Messenger.OnCondition(inoIoData.AcquisitionStatus.OfflineReason0 AND _onlineTimer.Q).Info('<#Camera offline:The vision system$'s job is being modified.#>');
Messenger.OnCondition(inoIoData.AcquisitionStatus.OfflineReason0 AND _onlineTimer.Q).Info('<#Camera offline:A discrete signal is holding the vision system Offline.#>');
Messenger.OnCondition(inoIoData.AcquisitionStatus.OfflineReason0 AND _onlineTimer.Q).Info('<#Camera offline:A communications protocol is holding the vision system Offline.#>');
END_METHOD

METHOD INTERNAL InvalidReference : BOOL
InvalidReference := FALSE;
IF NOT __ISVALIDREF(inoIoData) THEN
	_varInfo :=__VARINFO(inoIoData);
	Messenger.Programming(_sb.Clear().Append('<#Invalid reference: #>').Append(_varInfo.Symbol).ToString());
    InvalidReference := TRUE;
END_IF
END_METHOD

PROPERTY LastResultData : TcoInsightResults_v_5_x_x
GET
LastResultData := THIS^._results;
END_GET
END_PROPERTY

(*~
	<docu>
		<summary>
			Restores this instance to the Ready state. Can be called explicitly or from within one of the restore mechanisms.	
		</summary>			
	</docu>	
~*)
METHOD Restore : ITcoRestorable
_updateSignalStatesTask.Restore();
_changeJobByNumberTask.Restore();
_changeJobByNameTask.Restore();
_clearInspectionResultsTask.Restore();
_softEventTask.Restore();
_triggerTask.Restore();
_clearUserDataTask.Restore();
_setUserDataTask.Restore();

Tc2_System.MEMSET(destAddr:= ADR(THIS^._results.InspectionResults) , fillByte:= 0 , n:= SIZEOF(THIS^._results.InspectionResults));
Tc2_System.MEMSET(destAddr:= ADR(THIS^._userData.UserData) , fillByte:= 0 , n:= SIZEOF(THIS^._userData.UserData));


THIS^._results.InspectionId := 0;
THIS^._results.ResultCode := 0;
	
IF InvalidReference() THEN
    RETURN;
END_IF

Tc2_System.MEMSET(destAddr:= ADR(THIS^.inoIoData) , fillByte:= 0 , n:= SIZEOF(THIS^.inoIoData));

_status.ActionDescription := '<#Restore executed!#>';
_restoreTask.Restore();
END_METHOD

(*~
	<docu>
		<summary>
		    Custom service (manual, maintenance) logic.
			This method must be implemented in derived class.
		</summary>			
	</docu>	
~*)
METHOD PROTECTED ServiceMode
END_METHOD

(*~
	<docu>
		<summary>
			Set user data. 		
		</summary>			
	</docu>	
~*)
METHOD SetUserData : TcoCore.ITcoTaskStatus
SetUserData := THIS^._setUserDataTask.Invoke();
END_METHOD

METHOD SetUserDataAsByte : BOOL;
VAR_INPUT
	inValue : BYTE;
	inPosition : UINT;	
END_VAR
VAR
	_bufferSize : UINT; 
	_size : UINT; 
END_VAR
SetUserDataAsByte := FALSE;

_size := SIZEOF(inValue);

_bufferSize := SIZEOF(THIS^._userData.UserData)/SIZEOF(THIS^._userData.UserData[0]);

IF (inPosition +_size) > THIS^._config.UserDataSize THEN
	Messenger.Info('<#Index of UserData in method SetUserDataAsByte exceeds the size hardware structure mapped#>');
	RETURN;
END_IF

IF (inPosition +_size) > _bufferSize THEN
	Messenger.Info('<#Index of UserData in method SetUserDataAsByte exceeds the defined size#>');
	RETURN;
END_IF

THIS^._userData.UserData[inPosition]:=inValue;

SetUserDataAsByte := TRUE;
END_METHOD

METHOD SetUserDataAsDint : BOOL
VAR_INPUT
	inValue : DINT;
	inPosition : UINT;	
END_VAR
VAR
	_index : UINT;
	_size : UINT;
	_bufferSize : UINT; 
END_VAR
SetUserDataAsDint := FALSE;

_size := SIZEOF(inValue);

_bufferSize := SIZEOF(THIS^._userData.UserData)/SIZEOF(THIS^._userData.UserData[0]);

IF (inPosition +_size) > THIS^._config.UserDataSize THEN
	Messenger.Info('<#Index of UserData in method SetUserDataAsDint exceeds the size hardware structure mapped#>');
	RETURN;
END_IF

IF (inPosition +_size) > _bufferSize THEN
	Messenger.Info('<#Index of UserData in method SetUserDataAsDint exceeds the defined size#>');
	RETURN;
END_IF

TcoDintToBytes(THIS^._config.DataFormat,
				inValue,
				_userData.UserData[inPosition],
				_userData.UserData[inPosition+1],
				_userData.UserData[inPosition+2],
				_userData.UserData[inPosition+3]);	

SetUserDataAsDint := TRUE;
END_METHOD

METHOD SetUserDataAsReal : BOOL
VAR_INPUT
	inValue : DINT;
	inPosition : UINT;	
END_VAR
VAR
	_index : UINT;
	_size : UINT;
	_bufferSize : UINT; 
END_VAR
SetUserDataAsReal := FALSE;

_size := SIZEOF(inValue);

_bufferSize := SIZEOF(THIS^._userData.UserData)/SIZEOF(THIS^._userData.UserData[0]);

IF (inPosition +_size) > THIS^._config.UserDataSize THEN
	Messenger.Info('<#Index of UserData in method SetUserDataAsReal exceeds the size hardware structure mapped#>');
	RETURN;
END_IF

IF (inPosition +_size) > _bufferSize THEN
	Messenger.Info('<#Index of UserData in method SetUserDataAsReal exceeds the defined size#>');
	RETURN;
END_IF

	
TcoRealToBytes(THIS^._config.DataFormat,
				inValue,
				_userData.UserData[inPosition],
				_userData.UserData[inPosition+1],
				_userData.UserData[inPosition+2],
				_userData.UserData[inPosition+3]);			

SetUserDataAsReal := TRUE;
END_METHOD

METHOD SetUserDataAsString : BOOL
VAR_INPUT
	inValue : STRING;
	inPosition : UINT;	
END_VAR
VAR
	_index : UINT;
	_size : UINT;
	_bufferSize : UINT; 
END_VAR
SetUserDataAsString := FALSE;

_size := LEN(inValue);

_bufferSize := SIZEOF(THIS^._userData.UserData)/SIZEOF(THIS^._userData.UserData[0]);

IF (inPosition +_size) > THIS^._config.UserDataSize THEN
	Messenger.Info('<#Index of UserData in method SetUserDataAsString exceeds the size hardware structure mapped#>');
	RETURN;
END_IF

IF (inPosition +_size) > _bufferSize THEN
	Messenger.Info('<#Index of UserData in method SetUserDataAsString exceeds the defined size#>');
	RETURN;
END_IF

FOR	_index := 1 TO _size BY 1 DO	
	_userData.UserData[inPosition + _index-1] := F_ToASC(MID(inValue,1,_index));
END_FOR;

FOR	_index := inPosition +_size TO _bufferSize BY 1 DO	
	_userData.UserData[_index] := 0;
END_FOR;

SetUserDataAsString := TRUE;
END_METHOD

(*~
	<docu>
		<summary>
			Gets the `SetUserDataTask` task that controls to set of the user data. 		
		</summary>			
	</docu>	
~*)
PROPERTY SetUserDataTask : TcoCore.ITcoTaskStatus
GET
SetUserDataTask := THIS^._setUserDataTask;
END_GET
END_PROPERTY

(*~
	<docu>
		<summary>
			Executes the soft event. 		
		</summary>			
	</docu>	
~*)
METHOD SoftEvent : TcoCore.ITcoTaskStatus
VAR_INPUT
    inSoftEventNumber : UINT;
END_VAR
SoftEvent := THIS^._softEventTask.InvokeWithParameters(inSoftEventNumber);
END_METHOD

(*~
	<docu>
		<summary>
			Gets the `ClearResultDataTask` task that controls clearing of the results data. 		
		</summary>			
	</docu>	
~*)
PROPERTY SoftEventTask : TcoCore.ITcoTaskStatus
GET
SoftEventTask := THIS^._softEventTask;
END_GET
END_PROPERTY

(*~
	<docu>
		<summary>
			Gets the status of the sensor. 					
		</summary>			
	</docu>	
~*)
PROPERTY Status : REFERENCE TO TcoInsightStatus_v_5_x_x
GET
Status REF= _status;
END_GET
END_PROPERTY

(*~
	<docu>
		<summary>
			Triggers the reading sequence and waits for results. 		
		</summary>			
	</docu>	
~*)
METHOD Trigger : TcoCore.ITcoTaskStatus
Trigger := THIS^._triggerTask.Invoke();
END_METHOD

(*~
	<docu>
		<summary>
			Gets the `TriggerTask` result. 		
		</summary>			
	</docu>	
~*)
PROPERTY TriggerTask : TcoCore.ITcoTaskStatus
GET
TriggerTask := THIS^._triggerTask;
END_GET
END_PROPERTY

METHOD INTERNAL UpdateSignalStates
_status.SignalStatus.AcquisitionTriggerEnable := inoIoData.AcquisitionControl.AcquisitionTriggerEnable;
_status.SignalStatus.AcquisitionTrigger := inoIoData.AcquisitionControl.AcquisitionTrigger;
_status.SignalStatus.ClearExposureComplete := inoIoData.AcquisitionControl.ClearExposureComplete;
_status.SignalStatus.SetOffline := inoIoData.AcquisitionControl.SetOffline;
  
_status.SignalStatus.EnableResultsBuffering := inoIoData.InspectionControl.EnableResultsBuffering;
_status.SignalStatus.AcknowledgeInspectionResults := inoIoData.InspectionControl.AcknowledgeInspectionResults;
_status.SignalStatus.ExtendedUserDataSet := inoIoData.InspectionControl.ExtendedUserDataSet;
_status.SignalStatus.ExecuteCommand := inoIoData.InspectionControl.ExecuteCommand;
_status.SignalStatus.ClearError := inoIoData.InspectionControl.ClearError;
  
_status.SignalStatus.Command := inoIoData.CommandControl.Command;
  
_status.SignalStatus.TriggerSoftEvent.0 := inoIoData.SoftEventControl.TriggerSoftEvent[0];
_status.SignalStatus.TriggerSoftEvent.1 := inoIoData.SoftEventControl.TriggerSoftEvent[1];
_status.SignalStatus.TriggerSoftEvent.2 := inoIoData.SoftEventControl.TriggerSoftEvent[2];
_status.SignalStatus.TriggerSoftEvent.3 := inoIoData.SoftEventControl.TriggerSoftEvent[3];
_status.SignalStatus.TriggerSoftEvent.4 := inoIoData.SoftEventControl.TriggerSoftEvent[4];
_status.SignalStatus.TriggerSoftEvent.5 := inoIoData.SoftEventControl.TriggerSoftEvent[5];
_status.SignalStatus.TriggerSoftEvent.6 := inoIoData.SoftEventControl.TriggerSoftEvent[6];
_status.SignalStatus.TriggerSoftEvent.7 := inoIoData.SoftEventControl.TriggerSoftEvent[7];
	
_status.SignalStatus.AcquisitionTriggerReady := inoIoData.AcquisitionStatus.AcquisitionTriggerReady;
_status.SignalStatus.AcquisitionTriggerAcknowledge := inoIoData.AcquisitionStatus.AcquisitionTriggerAcknowledge;
_status.SignalStatus.ExposureComplete := inoIoData.AcquisitionStatus.ExposureComplete;
_status.SignalStatus.MissedAcquisition := inoIoData.AcquisitionStatus.MissedAcquisition;
_status.SignalStatus.OfflineReason0 := inoIoData.AcquisitionStatus.OfflineReason0;
_status.SignalStatus.OfflineReason1 := inoIoData.AcquisitionStatus.OfflineReason1;
_status.SignalStatus.OfflineReason2 := inoIoData.AcquisitionStatus.OfflineReason2;
_status.SignalStatus.Online := inoIoData.AcquisitionStatus.Online;
_status.SignalStatus.AcquisitionID := inoIoData.AcquisitionStatus.AcquisitionID;

_status.SignalStatus.SystemBusy := inoIoData.InspectionStatus.SystemBusy;
_status.SignalStatus.InspectionCompleted := inoIoData.InspectionStatus.InspectionCompleted;
_status.SignalStatus.ResultsBufferOverrun := inoIoData.InspectionStatus.ResultsBufferOverrun;
_status.SignalStatus.ResultsValid := inoIoData.InspectionStatus.ResultsValid;
_status.SignalStatus.CommandExecuting := inoIoData.InspectionStatus.CommandExecuting;
_status.SignalStatus.CommandComplete := inoIoData.InspectionStatus.CommandComplete;
_status.SignalStatus.CommandFailed := inoIoData.InspectionStatus.CommandFailed;
_status.SignalStatus.ExtendedUserDataSetAcknowledge := inoIoData.InspectionStatus.ExtendedUserDataSetAcknowledge;
_status.SignalStatus.OverallJobPassFail := inoIoData.InspectionStatus.OverallJobPassFail;
_status.SignalStatus.TestRunReady := inoIoData.InspectionStatus.TestRunReady;
_status.SignalStatus.Error := inoIoData.InspectionStatus.Error;
_status.SignalStatus.ErrorCode := inoIoData.InspectionStatus.ErrorCode;

_status.SignalStatus.CurrentJobID := inoIoData.CommandControl.CurrentJobID;

_status.SignalStatus.TriggerSoftEventAcknowledge.0 := inoIoData.SoftEventControl.TriggerSoftEventAcknowledge[0];
_status.SignalStatus.TriggerSoftEventAcknowledge.1 := inoIoData.SoftEventControl.TriggerSoftEventAcknowledge[1];
_status.SignalStatus.TriggerSoftEventAcknowledge.2 := inoIoData.SoftEventControl.TriggerSoftEventAcknowledge[2];
_status.SignalStatus.TriggerSoftEventAcknowledge.3 := inoIoData.SoftEventControl.TriggerSoftEventAcknowledge[3];
_status.SignalStatus.TriggerSoftEventAcknowledge.4 := inoIoData.SoftEventControl.TriggerSoftEventAcknowledge[4];
_status.SignalStatus.TriggerSoftEventAcknowledge.5 := inoIoData.SoftEventControl.TriggerSoftEventAcknowledge[5];
_status.SignalStatus.TriggerSoftEventAcknowledge.6 := inoIoData.SoftEventControl.TriggerSoftEventAcknowledge[6];
_status.SignalStatus.TriggerSoftEventAcknowledge.7 := inoIoData.SoftEventControl.TriggerSoftEventAcknowledge[7];

_status.SignalStatus.InspectionID := inoIoData.ResultsData.InspectionID;
_status.SignalStatus.ResultCode := inoIoData.ResultsData.ResultCode;

_updateSignalStatesTask.DoneWhen(TRUE);
END_METHOD

PROPERTY UserData : TcoInsightUser_v_5_x_x
GET
UserData := _userData;
END_GET
END_PROPERTY

END_FUNCTION_BLOCK
